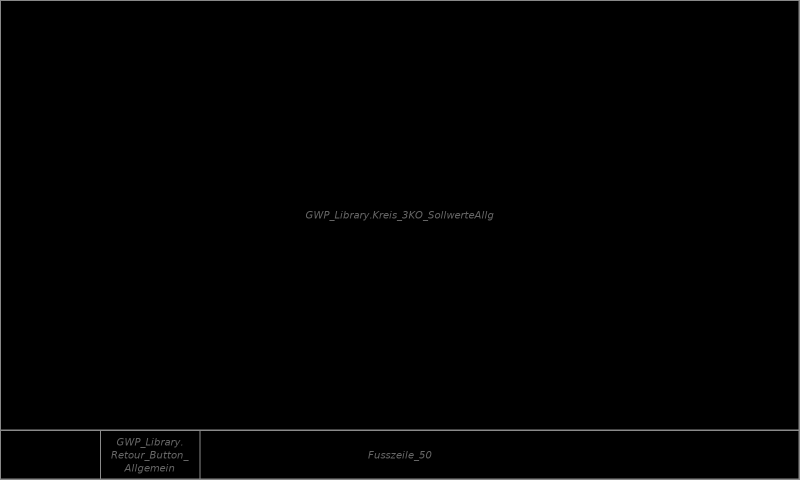
VISUALIZATION Kreis_3KO_SollwerteAllg  // 800x480
    Frame (0,0 800x430)
        shows GWP_Library.Kreis_3KO_SollwerteAllg(FB_Kreis_3KO := Main.Kreis_3KO_0)
    Group (0,430 800x50)
        Frame (0,0 800x50)
            shows Fusszeile_50()
        Frame (100,0 100x50)
            shows GWP_Library.Retour_Button_Allgemein()
END_VISUALIZATION

(* stored: Version 1.1.0.1, ProductVersion 3.1.4022.6
   Visu Kreis_3KO_SollwerteAllg: Id {be13ebbd-385a-49ce-bd6d-e2341d01c7d7} *)
